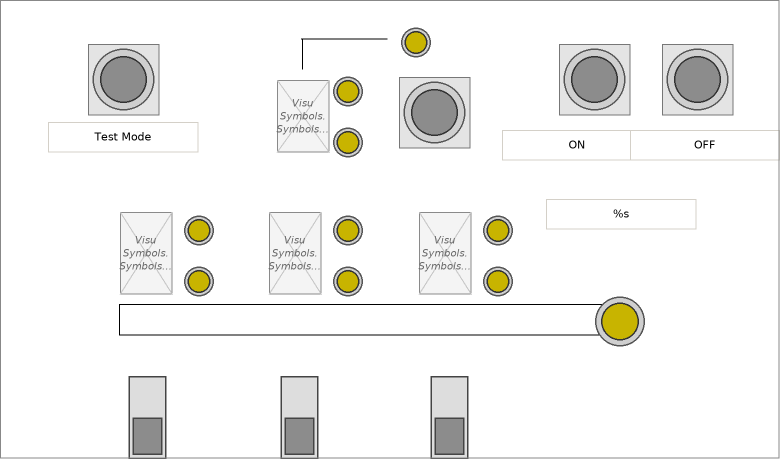
VISUALIZATION Visualization  // 780x459
    Rectangle (119,304 492x31)
    Lamp1 (577,293 86x57), variable: Hmi_Data_Exchange.bConveyorIsRunning, style: Lamp-Lamp1-Yellow
    Lamp1 (182,261 34x41), variable: Hmi_Data_Exchange.bInfeedCylinderRetract, style: Lamp-Lamp1-Yellow
    Lamp1 (182,210 34x41), variable: Hmi_Data_Exchange.bInfeedCylinderExtend, style: Lamp-Lamp1-Yellow
    Lamp1 (331,261 34x41), variable: Hmi_Data_Exchange.bTesterStopperCylinderRetract, style: Lamp-Lamp1-Yellow
    Lamp1 (331,210 34x41), variable: Hmi_Data_Exchange.bTesterStopperCylinderExtend, style: Lamp-Lamp1-Yellow
    Lamp1 (481,261 34x41), variable: Hmi_Data_Exchange.bKickerCylinderRetract, style: Lamp-Lamp1-Yellow
    Lamp1 (481,210 34x41), variable: Hmi_Data_Exchange.bKickerCylinderExtend, style: Lamp-Lamp1-Yellow
    Lamp1 (331,122 34x41), variable: Hmi_Data_Exchange.bTesterHeadCylinderExtend, style: Lamp-Lamp1-Yellow
    Lamp1 (331,71 34x41), variable: Hmi_Data_Exchange.bTesterHeadCylinderRetract, style: Lamp-Lamp1-Yellow
    Image (120,212 52x82), invisible if: NOT Hmi_Data_Exchange.bInfeedCylinderProductVisible, image: VisuSymbols.Symbols.ArrowBoldUp
    Image (269,212 52x82), invisible if: NOT Hmi_Data_Exchange.bTesterProductVisible, image: VisuSymbols.Symbols.ArrowBoldUp
    Image (419,212 52x82), invisible if: NOT Hmi_Data_Exchange.bKickerProductVisible, image: VisuSymbols.Symbols.ArrowBoldUp
    DipSwitch (105,376 85x83), variable: Hmi_Data_Exchange.bInfeedCylinderProductVisible, behaviour: TOGGLE, style: Switch-DipSwitch-Gray
    DipSwitch (257,376 85x83), variable: Hmi_Data_Exchange.bTesterProductVisible, behaviour: TOGGLE, style: Switch-DipSwitch-Gray
    DipSwitch (407,376 85x83), variable: Hmi_Data_Exchange.bKickerProductVisible, behaviour: TOGGLE, style: Switch-DipSwitch-Gray
    PushSwitch (88,40 71x79), variable: Hmi_Data_Exchange.bTestMode, behaviour: TOGGLE, style: Switch-PushSwitch-Gray
    PushSwitch (559,40 71x79), variable: Hmi_Data_Exchange.bHmiControlOn, behaviour: TOGGLE, style: Switch-PushSwitch-Gray
    PushSwitch (662,40 71x79), variable: Hmi_Data_Exchange.bHmiControlOFF, behaviour: TOGGLE, style: Switch-PushSwitch-Gray
    Image (277,80 52x72), image: VisuSymbols.Symbols.ArrowBoldDown
    Lamp1 (399,22 34x41), variable: Hmi_Data_Exchange.bAirTestPressureValve, style: Lamp-Lamp1-Yellow
    Line (387,39) (301,39)
    Line (302,39) (302,69)
    Textfield (502,130 150x30), "ON"
    Textfield (630,130 150x30), "OFF"
    Textfield (48,122 150x30), "Test Mode"
    Textfield (546,199 150x30), "%s", text variable: Hmi_Data_Exchange.eCurrentStep
    PushSwitch (399,73 71x79), variable: Hmi_Data_Exchange.bBottleQualityOk, behaviour: TOGGLE, style: Switch-PushSwitch-Gray
END_VISUALIZATION

(* stored: Version 1.1.0.1
   Visu Visualization: Id {df45bad7-bbb7-4704-b69a-82f20166bf80} *)
